SUBAPPLICATION mapping_Softkeys (* Subapplication Type *)
  (* Standard: 61499-2 *)
  (* Version 1.0, 2023-01-29, Franz *)
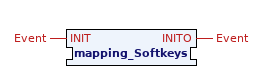
  EVENT_INPUT
    INIT;
  END_EVENT
  EVENT_OUTPUT
    INITO;
  END_EVENT
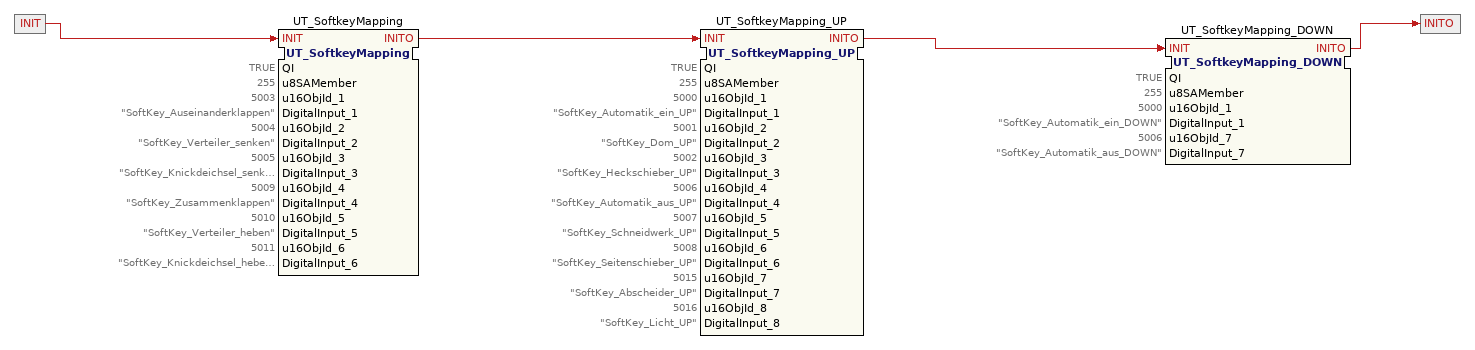
  FBS
    UT_SoftkeyMapping : UT_SoftkeyMapping(QI := TRUE, u8SAMember := 255, u16ObjId_1 := 5003, DigitalInput_1 := "SoftKey_Auseinanderklappen", u16ObjId_2 := 5004, DigitalInput_2 := "SoftKey_Verteiler_senken", u16ObjId_3 := 5005, DigitalInput_3 := "SoftKey_Knickdeichsel_senken", u16ObjId_4 := 5009, DigitalInput_4 := "SoftKey_Zusammenklappen", u16ObjId_5 := 5010, DigitalInput_5 := "SoftKey_Verteiler_heben", u16ObjId_6 := 5011, DigitalInput_6 := "SoftKey_Knickdeichsel_heben");
    UT_SoftkeyMapping_UP : UT_SoftkeyMapping_UP(QI := TRUE, u8SAMember := 255, u16ObjId_1 := 5000, DigitalInput_1 := "SoftKey_Automatik_ein_UP", u16ObjId_2 := 5001, DigitalInput_2 := "SoftKey_Dom_UP", u16ObjId_3 := 5002, DigitalInput_3 := "SoftKey_Heckschieber_UP", u16ObjId_4 := 5006, DigitalInput_4 := "SoftKey_Automatik_aus_UP", u16ObjId_5 := 5007, DigitalInput_5 := "SoftKey_Schneidwerk_UP", u16ObjId_6 := 5008, DigitalInput_6 := "SoftKey_Seitenschieber_UP", u16ObjId_7 := 5015, DigitalInput_7 := "SoftKey_Abscheider_UP", u16ObjId_8 := 5016, DigitalInput_8 := "SoftKey_Licht_UP");
    UT_SoftkeyMapping_DOWN : UT_SoftkeyMapping_DOWN(QI := TRUE, u8SAMember := 255, u16ObjId_1 := 5000, DigitalInput_1 := "SoftKey_Automatik_ein_DOWN", u16ObjId_7 := 5006, DigitalInput_7 := "SoftKey_Automatik_aus_DOWN");
  END_FBS
  EVENT_CONNECTIONS
    INIT TO UT_SoftkeyMapping.INIT;
    UT_SoftkeyMapping.INITO TO UT_SoftkeyMapping_UP.INIT;
    UT_SoftkeyMapping_UP.INITO TO UT_SoftkeyMapping_DOWN.INIT;
    UT_SoftkeyMapping_DOWN.INITO TO INITO;
  END_CONNECTIONS
END_SUBAPPLICATION
